PROGRAM prgComEffIO
VAR
	fbCom		: FB_MqttCommunicator_V3;
END_VAR

fbCom(
	bConnect:= TRUE, 
	strAuthKey:=  'BMS99299754422' , 
	sUserName:= '9c801c0d-8c2c-4278-a890-f6835690b001', 
	sUserPassword:= '4eabb1b6-b62b-40a2-976a-790462614f0c', 
	eSavePositionCertificate:= eSavePositionOnPLC.ePostionHardDisk, 
	time_HeartBeat_sec 		:= T#15S,
	bConnected=> , 
	bError=> , 
	hrErrorCode=> , 
	eConnectionState=> , 
	eErrorMessage_Out=> );
(* old
	sUserName:= '42ed263c-2a5f-4093-831d-18453bb20ab2', 
	sUserPassword:= '1dfb7dd2-4ea2-4174-bf5e-9fabdb42463b', 

	*)

END_PROGRAM

(* stored: Version 1.1.0.1, ProductVersion 3.1.4024.12
   POU prgComEffIO: Id {cbcd318b-bf51-484c-bcaa-d6efcdf43fe3}, SpecialFunc None *)
